Yaskawa INFORM job: clamp_planes_program.JBI

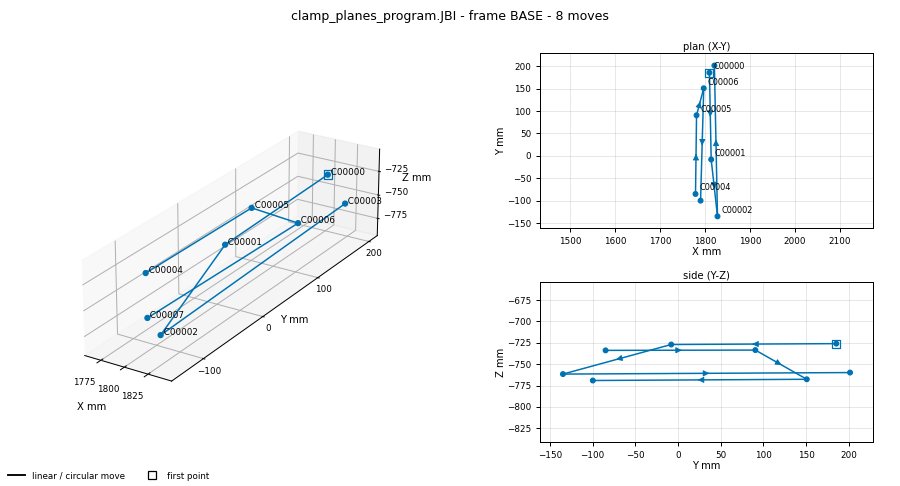
[picture p0: tool path of clamp_planes_program.JBI in frame BASE, 8 of 11 moves have a stored position in this frame; points joined in program order, loops and branches not executed]
/JOB
//NAME clamp_planes_program
//POS
///NPOS 8,0,8,0,0,0
///TOOL 0
///POSTYPE BASE
///RECTAN
///RCONF 0,0,0,0,0,0,0,0,0,0,0,0,0,0,0,0,0,0,0,0,0,0,0,0
C00000=1810.139647,185.264004,-725.990122,5.000000,-79.158186,175.000000
C00001=1814.029534,-7.928198,-727.020521,5.000000,-79.158186,175.000000
C00002=1828.057333,-134.614181,-761.614688,5.000000,-79.158186,175.000000
C00003=1821.183874,201.334835,-759.843795,180.000000,-60.000000,0.000000
C00004=1779.118034,-84.760702,-733.881447,5.000000,-76.181307,175.000000
C00005=1781.417586,90.531978,-733.524501,5.000000,-76.181307,175.000000
C00006=1797.417441,150.719908,-767.704555,5.000000,-76.181307,175.000000
C00007=1790.384446,-99.674657,-769.136365,180.000000,-60.000000,0.000000
///POSTYPE PULSE
///PULSE
EC00000=189440.0
EC00001=189440.0
EC00002=189440.0
EC00003=189440.0
EC00004=367616.0
EC00005=367616.0
EC00006=367616.0
EC00007=367616.0
//INST
///DATE 2023/08/16 17:15
///ATTR SC,RW,RJ
////FRAME BASE
///GROUP1 RB1,ST1
NOP
MOVJ P009 EX000 VJ=15.00
MOVJ C00000 EC00000 VJ=15.0
CALL JOB:SPYON
MOVL C00001 EC00001 V=150.0
MOVL C00002 EC00002 V=150.0
MOVL C00003 EC00003 V=150.0
CALL JOB:SPYOF
MOVJ P009 VJ=15.00
MOVJ C00004 EC00004 VJ=15.0
CALL JOB:SPYON
MOVL C00005 EC00005 V=150.0
MOVL C00006 EC00006 V=150.0
MOVL C00007 EC00007 V=150.0
CALL JOB:SPYOF
MOVJ P009 VJ=15.00
END
